PROGRAM PG_AddData
VAR
	i:UDINT;
	repeatTimer:TON;
	
	
	AlarmHistoryData_Write:ST_AlarmInfo_DB_save;
	ProductionHistoryData_Write:ST_Production_History_DB_Test;
	ProductionReport_Write:ST_OEE_ProductionReport;
	ProductionSummary_Write:ST_OEE_ProductionSummary;
	SoDuration_Write:ST_SoDuration;
	StopCount_Write:ST_StopCount;
	RegularCheckResults_Write:ST_RegularCheck_Results_DB;
	
	
	writeFailCount:UDINT;
	writeFailCount2:UDINT;
	writeFailCount3:UDINT;
	writeFailCount4:UDINT;
	writeFailCount5:UDINT;
	writeFailCount6:UDINT;
	writeFailCount7:UDINT;
END_VAR


//simulate that Peak Data amount as 500 ms
repeatTimer(IN:=TRUE,PT:=T#300MS);

IF repeatTimer.Q THEN
	
	repeatTimer(in:=FALSE);
	
	//simulate Peak save data amount
	FOR i:=0 TO GVL.Max_IndexNum-1 DO
		(*
		IF GVL.fbDataToNovRam[i].M_AlarmHistory(addData:=AlarmHistoryData_Write) = FALSE THEN
			writeFailCount:=writeFailCount+1;
		END_IF
		*)
		(*
		IF GVL.fbDataToNovRam[i].M_ProductionHistory(addData:=ProductionHistoryData_Write) = FALSE THEN
			writeFailCount2:=writeFailCount2+1;
		END_IF
		*)
		//(*
		IF GVL.fbDataToNovRam[i].M_ProductionReport(addData:=ProductionReport_Write) = FALSE THEN
			writeFailCount3:=writeFailCount3+1;
		END_IF
		//*)
		(*
		//write to db failed
		IF GVL.fbDataToNovRam[i].M_ProductionSummary(addData:=ProductionSummary_Write) = FALSE THEN
			writeFailCount4:=writeFailCount4+1;
		END_IF
		*)
		(*
		//write to db failed
		IF GVL.fbDataToNovRam[i].M_SoDuration(addData:=SoDuration_Write) = FALSE THEN
			writeFailCount5:=writeFailCount5+1;
		END_IF
		*)
		(*
		//Failed 需要faamid
		IF GVL.fbDataToNovRam[i].M_StopCount(addData:=StopCount_Write) = FALSE THEN
			writeFailCount6:=writeFailCount6+1;
		END_IF
		*)
		(*
		IF GVL.fbDataToNovRam[i].M_RegularCheckResults(addData:=RegularCheckResults_Write) = FALSE THEN
			writeFailCount7:=writeFailCount7+1;
		END_IF
		*)
	END_FOR
	
END_IF

END_PROGRAM

(* stored: Version 1.1.0.1, ProductVersion 3.1.4024.11
   POU PG_AddData: Id {54f410b2-b83a-4d7a-938e-1ab226b5f3f6}, SpecialFunc None *)
